FUNCTION F_Concat3 : STRING(255)
VAR_INPUT
	String1 : STRING(255);
	String2 : STRING(255);
	String3 : STRING(255);
END_VAR
VAR
END_VAR

F_Concat3 := CONCAT(String1,CONCAT(String2,String3));

END_FUNCTION

(* stored: Version 1.1.0.1, ProductVersion 3.1.4022.16
   POU F_Concat3: Id {84013d23-288a-4fb4-950b-8368975b8420}, SpecialFunc None *)
